FUNCTION_BLOCK E_CTD
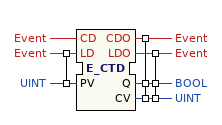
  EVENT_INPUT
    CD;
    LD WITH PV;
  END_EVENT
  EVENT_OUTPUT
    CDO WITH Q, CV;
    LDO WITH Q, CV;
  END_EVENT
  VAR_INPUT
    PV : UINT;
  END_VAR
  VAR_OUTPUT
    Q : BOOL;
    CV : UINT;
  END_VAR
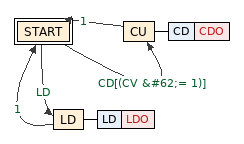
  EC_STATES
    START;
    CU : CD -> CDO;
    LD : LD -> LDO;
  END_STATES
  EC_TRANSITIONS
    START TO CU := CD[(CV &#62;= 1)];
    CU TO START := 1;
    START TO LD := LD;
    LD TO START := 1;
  END_TRANSITIONS
  ALGORITHM CD IN ST:
CV := CV - 1;&#38;#10;Q := (CV &#60;= 0);&#38;#10;
  END_ALGORITHM
  ALGORITHM LD IN ST:
CV := PV;&#38;#10;Q := (CV &#60;= 0);&#38;#10;
  END_ALGORITHM
END_FUNCTION_BLOCK
